DATA_BLOCK DB 810
TITLE =
AUTHOR : CB
STRUCT
WORD0 : WORD;	//
WORD1 : WORD;	//
WORD2 : WORD;	//
WORD3 : WORD;	//
END_STRUCT;
BEGIN
END_DATA_BLOCK
